// TwinCAT 3 PLC project FMTime
// Title: FM Time
// Company: FrameworkMonorepo
// ProjectVersion: 0.0.1
// ProgramVersion: 3.1.4024.0
// libraries:
//   FM Common Interfaces, * (FrameworkMonorepo)
//   FM Strings, * (FrameworkMonorepo)
//   Tc2_Standard, * (Beckhoff Automation GmbH)
//   Tc2_Utilities, * (Beckhoff Automation GmbH)
// project tree:
//   Clocks/ Clock.TcPOU, PeriodicTrigger.TcPOU
//   Convert/ SecondsToTime.TcPOU, TimeToSeconds.TcPOU
//   CycleTime/ GetCycleTimeInSeconds.TcPOU
//   TimeProvider/ TimeProvider.TcPOU
//   Version/ Global_Version.TcGVL
// (motion and I/O tree: see PLC project fmtypes)
// real-time tasks:
//   TASK BindingTestTask: cycle T#1ms, priority 20, ADS port 350
//   TASK PlcTask: cycle T#1ms, priority 21, ADS port 351
//   TASK PlcTask1: cycle T#1ms, priority 22, ADS port 352
//   TASK PlcTask2: cycle T#1ms, priority 23, ADS port 353
//   TASK MathTestTask: cycle T#1ms, priority 24, ADS port 354
//   TASK TimesTestsTask: cycle T#1ms, priority 25, ADS port 355

// ---- Version/Global_Version.TcGVL
{attribute 'TcGenerated'}
{attribute 'no-analysis'}
{attribute 'linkalways'}
// This function has been automatically generated from the project information.
VAR_GLOBAL CONSTANT
	{attribute 'const_non_replaced'}
	stLibVersion_FM_Time : ST_LibVersion := (iMajor := 0, iMinor := 0, iBuild := 1, iRevision := 0, nFlags := 0, sVersion := '0.0.1');
END_VAR

// ---- Clocks/Clock.TcPOU
FUNCTION_BLOCK Clock IMPLEMENTS Cyclic
VAR
	_Enable : BOOL;
	_Period : TIME;
	_Duty : LREAL := 0.5;
	switchTime : TIME;
	timer : TON;
	_Clock : BOOL;
END_VAR

METHOD PRIVATE CalcSwitchTime
switchTime := LREAL_TO_TIME(TIME_TO_LREAL(_Period) * _Duty);
END_METHOD

{attribute 'monitoring' := 'call'}
PROPERTY Clock : BOOL
GET
Clock := _Clock;
END_GET
END_PROPERTY

METHOD Cyclic
timer(IN := _Enable, PT := _Period);
IF (timer.Q) THEN
	timer(IN := FALSE);
	timer(IN := TRUE);
END_IF
_Clock := _Enable AND timer.ET >= switchTime;
END_METHOD

{attribute 'monitoring' := 'call'}
PROPERTY Duty : LREAL
GET
Duty := _Duty;
END_GET
SET
_Duty := Duty;
CalcSwitchTime();
END_SET
END_PROPERTY

{attribute 'monitoring' := 'call'}
PROPERTY Enable : BOOL
GET
Enable := _Enable;
END_GET
SET
_Enable := Enable;
END_SET
END_PROPERTY

{attribute 'monitoring' := 'call'}
PROPERTY Frequency : LREAL
GET
IF (_Period > T#0S) THEN
	Frequency := 1000/TIME_TO_LREAL(_Period);
ELSE
	Frequency := 0;
END_IF
END_GET
SET
IF (Frequency > 0) THEN
	_Period := LREAL_TO_TIME(1000/Frequency);
ELSE
	_Period := T#0S;
END_IF
CalcSwitchTime();
END_SET
END_PROPERTY

{attribute 'monitoring' := 'call'}
PROPERTY Period : TIME
GET
Period := _Period;
END_GET
SET
_Period := Period;
CalcSwitchTime();
END_SET
END_PROPERTY

END_FUNCTION_BLOCK

// ---- Clocks/PeriodicTrigger.TcPOU
FUNCTION_BLOCK PeriodicTrigger IMPLEMENTS Cyclic
VAR
	_Enable : BOOL;
	_Period : TIME;
	_PulseAtStart : BOOL; // If TRUE, pulse is generated at start of period. If FALSE, pulse is generated after period finishes.
	
	_Trigger : BOOL;
	timer : TON;
	justEnabled : R_TRIG;
END_VAR

METHOD Cyclic
justEnabled(CLK := _Enable);
IF (justEnabled.Q AND _PulseAtStart) THEN
	_Trigger := TRUE;
	timer(IN := TRUE, PT := _Period);
END_IF

IF (_Enable) THEN
	IF (NOT justEnabled.Q) THEN
		_Trigger := FALSE;
	END_IF
	
	timer(IN := TRUE, PT := _Period);
	IF (timer.Q) THEN
		_Trigger := TRUE;
		timer(IN := FALSE);
		timer(IN := TRUE);
	END_IF
ELSE
	timer(IN := FALSE);
END_IF
END_METHOD

{attribute 'monitoring' := 'call'}
PROPERTY Enable : BOOL
GET
Enable := _Enable;
END_GET
SET
_Enable := Enable;
END_SET
END_PROPERTY

{attribute 'monitoring' := 'call'}
PROPERTY Period : TIME
GET
Period := _Period;
END_GET
SET
_Period := Period;
END_SET
END_PROPERTY

{attribute 'monitoring' := 'call'}
PROPERTY PulseAtStart : BOOL
GET
PulseAtStart := _PulseAtStart;
END_GET
SET
_PulseAtStart := PulseAtStart;
END_SET
END_PROPERTY

{attribute 'monitoring' := 'call'}
PROPERTY Trigger : BOOL
GET
//Trigger := edgeTrigger.Q AND _Enable;
Trigger := _Trigger AND _Enable;
END_GET
END_PROPERTY

END_FUNCTION_BLOCK

// ---- Convert/SecondsToTime.TcPOU
FUNCTION SecondsToTime : TIME
VAR_INPUT
	seconds : LREAL;
END_VAR

SecondsToTime := LREAL_TO_TIME(seconds * 1000);

END_FUNCTION

// ---- Convert/TimeToSeconds.TcPOU
FUNCTION TimeToSeconds : LREAL
VAR_INPUT
	t : TIME;
END_VAR

TimeToSeconds := TIME_TO_LREAL(t) * 0.001;

END_FUNCTION

// ---- CycleTime/GetCycleTimeInSeconds.TcPOU
FUNCTION GetCycleTimeInSeconds : LREAL
VAR CONSTANT
	DefaultCTUnit : LREAL := 0.0000001; // PlcTaskSystemInfo.CycleTime is in [100*ns]
END_VAR
VAR
	cycleTime : UDINT;
END_VAR

cycleTime := _TaskInfo[GETCURTASKINDEXEX()].CycleTime;
GetCycleTimeInSeconds := TO_LREAL(cycleTime) * DefaultCTUnit;

END_FUNCTION

// ---- TimeProvider/TimeProvider.TcPOU
FUNCTION_BLOCK TimeProvider IMPLEMENTS Cyclic
VAR
	localSystemTime : FB_LocalSystemTime;
	getTimeZoneInformation : FB_GetTimeZoneInformation;
    timeZoneInformation : ST_TimeZoneInformation;
    specificLocalTimeToFileTime : FB_TzSpecificLocalTimeToFileTime;
    fileTime : T_FILETIME;
    onZerothSecondLastCycle : BOOL;
END_VAR

METHOD Cyclic
VAR_INPUT
END_VAR
localSystemTime(bEnable := FALSE);

// On the zeroth second of each minute sync timezone information
IF (timeZoneInformation.standardName = '' OR (localSystemTime.systemTime.wSecond = 0 AND NOT onZerothSecondLastCycle)) THEN
    getTimeZoneInformation(sNetID := '', bExecute := TRUE, tzInfo => timeZoneInformation);
END_IF;

// Convert local system time to unix timestamps
specificLocalTimeToFileTime(in := Tc2_Utilities.SYSTEMTIME_TO_FILETIME(localSystemTime.systemTime), tzInfo := timeZoneInformation, out => fileTime);

onZerothSecondLastCycle := localSystemTime.systemTime.wSecond = 0;
END_METHOD

METHOD FB_init : BOOL
VAR_INPUT
	bInitRetains : BOOL; // if TRUE, the retain variables are initialized (warm start / cold start)
	bInCopyCode : BOOL;  // if TRUE, the instance afterwards gets moved into the copy code (online change)
END_VAR
localSystemTime(bEnable := TRUE);
END_METHOD

METHOD GetMonthName : STRING
VAR_INPUT
	monthNumber			: UINT;
	shortName			: BOOL;
END_VAR
IF shortName THEN
	CASE monthNumber OF
		1	: GetMonthName := 'Jan';
		2	: GetMonthName := 'Feb';
		3	: GetMonthName := 'Mar';
		4	: GetMonthName := 'Apr';
		5	: GetMonthName := 'May';
		6	: GetMonthName := 'Jun';
		7	: GetMonthName := 'Jul';
		8	: GetMonthName := 'Aug';
		9	: GetMonthName := 'Sep';
		10	: GetMonthName := 'Oct';
		11	: GetMonthName := 'Nov';
		12	: GetMonthName := 'Dec';
	END_CASE
ELSE
	CASE monthNumber OF
		1	: GetMonthName := 'January';
		2	: GetMonthName := 'February';
		3	: GetMonthName := 'March';
		4	: GetMonthName := 'April';
		5	: GetMonthName := 'May';
		6	: GetMonthName := 'June';
		7	: GetMonthName := 'July';
		8	: GetMonthName := 'August';
		9	: GetMonthName := 'September';
		10	: GetMonthName := 'October';
		11	: GetMonthName := 'November';
		12	: GetMonthName := 'December';
	END_CASE
END_IF
END_METHOD

METHOD GetTimeString : STRING
VAR_INPUT
	format : STRING; // Example: {hh}:{mm}:{ss}:{SSS} {dd}:{MM}:{yyyy} https://www.ibm.com/docs/en/rtw/9.0.1?topic=reference-formatting-parsing-date-time-patterns
END_VAR
VAR
	placeholder : STRING(4);
	
	beginIndex	: INT;
	endIndex	: INT;
	length		: INT;
		
END_VAR
GetTimeString := format;

WHILE (beginIndex := FIND(GetTimeString, '{')) > 0 AND (endIndex := FIND(GetTimeString, '}')) > (beginIndex + 1) AND  (length := endIndex - beginIndex - 1) > 0 DO
	
	placeholder := MID(STR := GetTimeString, POS := beginIndex + 1, LEN := length);
		
	IF 		placeholder = 'h' 		THEN GetTimeString := REPLACE( STR1 := GetTimeString, STR2 := TO_STRING(localSystemTime.systemTime.wHour), L := length + 2, P := beginIndex);
	ELSIF 	placeholder = 'hh' 		THEN GetTimeString := REPLACE( STR1 := GetTimeString, STR2 := AddLeadingZeros(TO_STRING(localSystemTime.systemTime.wHour), 2), L := length + 2, P := beginIndex);
	ELSIF 	placeholder = 'm' 		THEN GetTimeString := REPLACE( STR1 := GetTimeString, STR2 := TO_STRING(localSystemTime.systemTime.wMinute), L := length + 2, P := beginIndex);
	ELSIF 	placeholder = 'mm' 		THEN GetTimeString := REPLACE( STR1 := GetTimeString, STR2 := AddLeadingZeros(TO_STRING(localSystemTime.systemTime.wMinute), 2), L := length + 2, P := beginIndex);
	ELSIF 	placeholder = 's' 		THEN GetTimeString := REPLACE( STR1 := GetTimeString, STR2 := TO_STRING(localSystemTime.systemTime.wSecond), L := length + 2, P := beginIndex);
	ELSIF 	placeholder = 'ss' 		THEN GetTimeString := REPLACE( STR1 := GetTimeString, STR2 := AddLeadingZeros(TO_STRING(localSystemTime.systemTime.wSecond), 2), L := length + 2, P := beginIndex);
	ELSIF 	placeholder = 'S' 		THEN GetTimeString := REPLACE( STR1 := GetTimeString, STR2 := TO_STRING(localSystemTime.systemTime.wMilliseconds/100), L := length + 2, P := beginIndex);
	ELSIF 	placeholder = 'SS' 		THEN GetTimeString := REPLACE( STR1 := GetTimeString, STR2 := AddLeadingZeros(TO_STRING(localSystemTime.systemTime.wMilliseconds/10), 2), L := length + 2, P := beginIndex);
	ELSIF 	placeholder = 'SSS' 	THEN GetTimeString := REPLACE( STR1 := GetTimeString, STR2 := AddLeadingZeros(TO_STRING(localSystemTime.systemTime.wMilliseconds), 3), L := length + 2, P := beginIndex);
	ELSIF 	placeholder = 'd' 		THEN GetTimeString := REPLACE( STR1 := GetTimeString, STR2 := TO_STRING(localSystemTime.systemTime.wDay), L := length + 2, P := beginIndex);
	ELSIF 	placeholder = 'dd' 		THEN GetTimeString := REPLACE( STR1 := GetTimeString, STR2 := AddLeadingZeros(TO_STRING(localSystemTime.systemTime.wDay), 2), L := length + 2, P := beginIndex);
	ELSIF 	placeholder = 'ddd' 	THEN GetTimeString := REPLACE( STR1 := GetTimeString, STR2 := GetWeekdayName(localSystemTime.systemTime.wDayOfWeek, TRUE), L := length + 2, P := beginIndex);
	ELSIF 	placeholder = 'dddd'	THEN GetTimeString := REPLACE( STR1 := GetTimeString, STR2 := GetWeekdayName(localSystemTime.systemTime.wDayOfWeek, FALSE), L := length + 2, P := beginIndex);
	ELSIF 	placeholder = 'M' 		THEN GetTimeString := REPLACE( STR1 := GetTimeString, STR2 := TO_STRING(localSystemTime.systemTime.wMonth), L := length + 2, P := beginIndex);
	ELSIF 	placeholder = 'MM' 		THEN GetTimeString := REPLACE( STR1 := GetTimeString, STR2 := AddLeadingZeros(TO_STRING(localSystemTime.systemTime.wMonth), 2), L := length + 2, P := beginIndex);
	ELSIF 	placeholder = 'MMM' 	THEN GetTimeString := REPLACE( STR1 := GetTimeString, STR2 := GetMonthName(localSystemTime.systemTime.wMonth, TRUE), L := length + 2, P := beginIndex);
	ELSIF 	placeholder = 'MMMM'	THEN GetTimeString := REPLACE( STR1 := GetTimeString, STR2 := GetMonthName(localSystemTime.systemTime.wMonth, FALSE), L := length + 2, P := beginIndex);
	ELSIF 	placeholder = 'y' OR placeholder = 'yy' OR placeholder = 'yyy' OR placeholder = 'yyyy'
									THEN GetTimeString := REPLACE( STR1 := GetTimeString, STR2 := RIGHT(TO_STRING(localSystemTime.systemTime.wYear), length), L := length + 2, P := beginIndex);
	ELSE 
			GetTimeString := REPLACE( STR1 := GetTimeString, STR2 := 'ERR', L := length + 2, P := beginIndex);
	END_IF
END_WHILE
END_METHOD

METHOD GetWeekdayName : STRING
VAR_INPUT
	weekDayNumber		: UINT;
	shortName			: BOOL;
END_VAR
IF shortName THEN
	CASE weekDayNumber OF
		0	: GetWeekdayName := 'Sun';
		1	: GetWeekdayName := 'Mon';
		2	: GetWeekdayName := 'Tue';
		3	: GetWeekdayName := 'Wed';
		4	: GetWeekdayName := 'Thu';
		5	: GetWeekdayName := 'Fri';
		6	: GetWeekdayName := 'Sat';
	END_CASE
ELSE
	CASE weekDayNumber OF
		0	: GetWeekdayName := 'Sunday';
		1	: GetWeekdayName := 'Monday';
		2	: GetWeekdayName := 'Tuesday';
		3	: GetWeekdayName := 'Wednesday';
		4	: GetWeekdayName := 'Thursday';
		5	: GetWeekdayName := 'Friday';
		6	: GetWeekdayName := 'Saturday';
	END_CASE
END_IF
END_METHOD

PROPERTY Timestamp : ULINT // Unix timestamp in milliseconds
GET
// TODO is this even right?
Timestamp := (SHL(DWORD_TO_ULINT(fileTime.dwHighDateTime), 32) + DWORD_TO_ULINT(fileTime.dwLowDateTime)) / 10000 - 11644473600000;
END_GET
END_PROPERTY

PROPERTY TimeStruct : TIMESTRUCT // Week starts with Sunday
GET
TimeStruct := localSystemTime.systemTime;
END_GET
END_PROPERTY

PROPERTY TimeStructISO8601 : TIMESTRUCT // Week starts with Monday
GET
TimeStructISO8601 := localSystemTime.systemTime;
IF TimeStructISO8601.wDayOfWeek = 0 THEN
	TimeStructISO8601.wDayOfWeek := 6; // Move Sunday to the end of the week
ELSE
	TimeStructISO8601.wDayOfWeek := TimeStructISO8601.wDayOfWeek - 1;
END_IF
END_GET
END_PROPERTY

END_FUNCTION_BLOCK
